// LS Electric XG5000 project: counter
// PLC NewPLC
// module base 0 slot 0: 입출력 모듈:XBC-DR20S (DC 24V 입력 12점, 릴레이 출력 8점)

PROGRAM NewProgram (task: 스캔 프로그램)

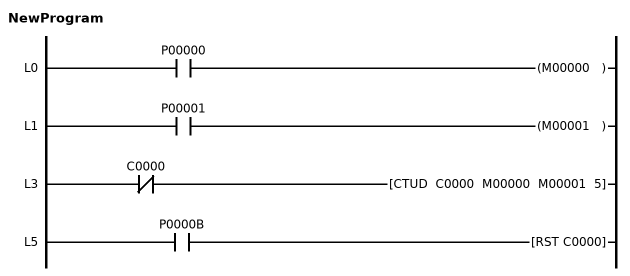
; L0
LOAD      P00000
OUT       M00000
; L1
LOAD      P00001
OUT       M00001
; L3
LOAD NOT  C0000
CTUD      C0000 M00000 M00001 5
; L5
LOAD      P0000B
RST       C0000